FUNCTION_BLOCK iCreateMgt (* Service Interface Function Block Type *)
  (* Standard: 61499-2 *)
  (* Version 0.0, 2012-08-15, 4DIAC-IDE, 4DIAC-Consortium *)
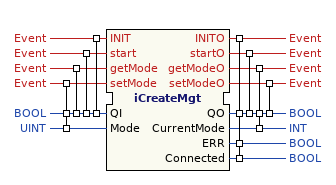
  EVENT_INPUT
    INIT WITH QI; (* INIT +(QI=T=1) Connect CBC to iRobot Create; INIT- (QI=F=0) disconnect *)
    start WITH QI; (* Puts Create into active mode (with motors) *)
    getMode WITH QI;
    setMode WITH Mode, QI;
  END_EVENT
  EVENT_OUTPUT
    INITO WITH QO, ERR, Connected; (* Initialization (+) or indication of service  (-) Confirm *)
    startO WITH QO; (* Indication from Resource *)
    getModeO WITH QO, CurrentMode;
    setModeO WITH QO;
  END_EVENT
  VAR_INPUT
    QI : BOOL; (* Event Input Qualifier *)
    Mode : UINT; (* Safe=0 safe, Passive=1 passive, Full=2 full, Off=3 *)
  END_VAR
  VAR_OUTPUT
    QO : BOOL; (* Event Output Qualifier *)
    CurrentMode : INT; (* Input data from resource *)
    ERR : BOOL; (* 0 if sucessful and a negative number if not *)
    Connected : BOOL;
  END_VAR
  SERVICE APPLICATION/RESOURCE (* Service Interface Function Block Type *)
    SEQUENCE normal_establishment
      APPLICATION.INIT+(PARAMS) -> APPLICATION.INITO+(PARAMS);
    END_SEQUENCE
    SEQUENCE unsuccessful_establishment
      APPLICATION.INIT+(PARAMS) -> APPLICATION.INITO-(STATUS);
    END_SEQUENCE
    SEQUENCE request_confirm
      APPLICATION.REQ+(SD) -> APPLICATION.CNF+(RD);
    END_SEQUENCE
    SEQUENCE request_inhibited
      APPLICATION.REQ-(SD) -> APPLICATION.CNF-(STATUS);
    END_SEQUENCE
    SEQUENCE request_error
      APPLICATION.REQ+(SD) -> APPLICATION.CNF-(STATUS);
    END_SEQUENCE
    SEQUENCE indication_response
      RESOURCE.indicate(RD) -> APPLICATION.IND+(RD);
      APPLICATION.RSP(QI,SD) -> RESOURCE.response(QI,SD);
    END_SEQUENCE
    SEQUENCE indication_inhibited
      RESOURCE.indicate(RD,QI=FALSE) -> RESOURCE.inhibited();
    END_SEQUENCE
    SEQUENCE error_indication
      RESOURCE.error(STATUS) -> APPLICATION.IND-(STATUS);
    END_SEQUENCE
    SEQUENCE application_initiated_termination
      APPLICATION.INIT-() -> APPLICATION.INITO-(STATUS);
    END_SEQUENCE
    SEQUENCE resource_initiated_termination
      -> APPLICATION.INITO-(STATUS);
    END_SEQUENCE
  END_SERVICE
END_FUNCTION_BLOCK
